Staubli VAL3: load.pgx

public program load(string x_sItem, num& x_nResult)
  local string l_sType
  local string l_sMessage
  local num i
  local num l_nResult
begin
  // load the select trajectory..already loaded
  call getTrajType(l_sType)
  if find(pt:libPath(),saveData:sPathTraj)==-1
    l_nResult=pt:libLoad(saveData:sPathTraj+l_sType)
    delay(0)
    if saveData:bDebug or l_nResult!=0
      ? "loading PALLET..."+saveData:sPathTraj+l_sType + toString("",l_nResult)
    endIf
  endIf
  // use the type...
  if isDefined(pt:tTraj[x_sItem])
    call pt:link_all(x_sItem)
    pEditPoint=pt:tTraj[x_sItem]
    pEditPoint.sID=x_sItem
    link(pEditPoint.fReference,world)
    link(pEditPoint.fFrame,pEditPoint.fReference)
  elseIf x_sItem!=""
    // not FOUND
    call language:message(l_sMessage,-7)
    x_nResult=-1
    popUpMsg(l_sMessage+x_sItem)
    pEditPoint.sID=""
  endIf
end
